FUNCTION flip_byte :  REAL
VAR_INPUT
	
	byte_array : ARRAY[0..3] OF BYTE;
END_VAR

VAR
		valor_flip : ARRAY[0..3] OF BYTE;
		pt: POINTER TO REAL;
		

		
END_VAR


//direcciones


valor_flip[0] := byte_array[3];
valor_flip[1] := byte_array[2];
valor_flip[2] := byte_array[1];
valor_flip[3] := byte_array[0];

pt := ADR(valor_flip);
flip_byte := pt^;

END_FUNCTION

(* stored: Version 1.1.0.1, ProductVersion 3.1.4024.4
   POU flip_byte: Id {9d098dce-4aa6-4ce4-9e2f-278a2ced4d6c}, SpecialFunc None *)
